TYPE ST_RobotParams :
STRUCT
    // ------------------------------------------------------------------
    // Dobot tuning parameters exchanged over TCP:6001. TCP is now the ONLY
    // robot channel -- start/stop moved from discrete I/O to STATE:n / CMD:n
    // frames (see nStateOut / nRobotCmd below). Field names and order match
    // the robot's SYNC string (see global.lua / dummy_server.py in
    // RobotBridge\Client_working_example). All INT so the classic VISU HMI
    // binds NumericInput directly. Defaults mirror the dummy server.
    // ------------------------------------------------------------------
    J_SPEED            : INT := 10;
    L_SPEED            : INT := 10;
    REPEATS            : INT := 2;
    START_WAIT         : INT := 500;
    WATER_WAIT         : INT := 500;
    STAND_WAIT         : INT := 2000;
    END_WAIT           : INT := 500;
    WATER_SPEED        : INT := 10;
    WAX_WAIT_TIME_IN   : INT := 500;
    WAX_WAIT_TIME_OUT  : INT := 500;
    WAX_SPEED          : INT := 10;

    // ------------------------------------------------------------------
    // Request flags -- FB_RobotTcpClient consumes each on the next idle
    // scan while Connected, sends the matching message, then auto-clears
    // the flag once the reply is received. Rising-level, not edge: setting
    // TRUE from the HMI is enough.
    // ------------------------------------------------------------------

    // Send GET_SYNC; the SYNC reply is parsed back into the 11 fields above.
    // The FB also raises this itself once, right after each (re)connect.
    bGetSync           : BOOL;

    // Send "sSetName:nSetVal" (e.g. "J_SPEED:15"); robot replies "OK: SET NAME".
    bSetParam          : BOOL;
    sSetName           : STRING(30);
    nSetVal            : INT;

    // Send "New_Bulb:1"; robot replies "OK: SET New_Bulb" and starts a fresh bulb.
    bTriggerNewBulb    : BOOL;

    // ------------------------------------------------------------------
    // State + command channel (replaces the retired discrete-I/O handshake).
    //
    // nStateOut : INT -- MAIN writes each scan. Value is TO_INT(eStep) in
    //   Automatic mode, or E_MasterAutoStep.MANUAL (30) when bAutoMode=FALSE.
    //   FB_RobotTcpClient sends "STATE:n" on change and every STATE_IDLE_MS
    //   as keep-alive.
    //
    // nRobotCmd : INT -- FB_RobotTcpClient writes each time a "CMD:n" reply
    //   arrives. MAIN R_TRIGs on nRobotCmd=1 (start cycle) and =2 (reset
    //   error). Robot is responsible for zeroing after the PLC's next state
    //   push acknowledges the command.
    // ------------------------------------------------------------------
    nStateOut          : INT;
    nRobotCmd          : INT;
END_STRUCT
END_TYPE

(* stored: Version 1.1.0.1, ProductVersion 3.1.4026.18
   DUT ST_RobotParams: Id {48e0cfb9-5ce6-4b32-9c93-d402e6dcbe42} *)
